RoboDK station: Ensamble.rdk

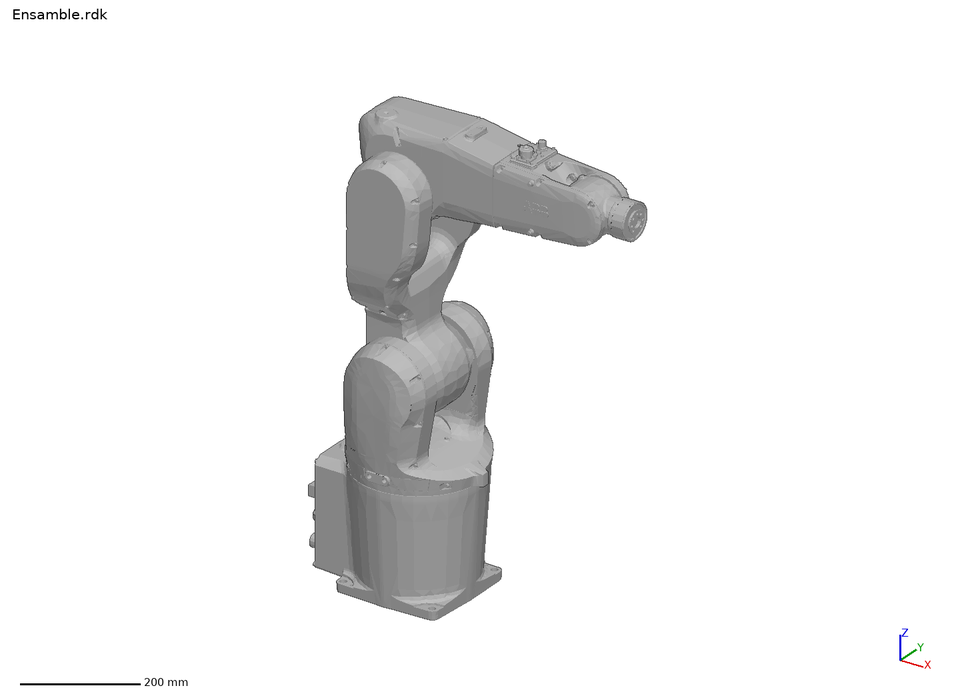
[picture v0: the station drawn from its stored meshes, robots at their saved joint values, targets as dots, program paths as lines]
Station Ensamble (saved by RoboDK 5.3.4). Poses are relative to the parent item; angles as X-Y-Z fixed-axis rotations.
  - object robot_irb_1200-7_0_7_01 at (0, 0, 0) mm, rotated rx 90 ry 0 rz 0 deg, size 285.2 x 192.7 x 127.5 mm, geometry from robot_irb_1200-7_0_7_01.STEP
  - object robot_irb_1200-7_0_7_02 at (0, 0, 0) mm, rotated rx 90 ry 0 rz 0 deg, size 5.5 x 44 x 44 mm, geometry from robot_irb_1200-7_0_7_02.STEP
  - object robot_irb_1200-7_0_7_03 at (0, 0, 0) mm, rotated rx 90 ry 0 rz 0 deg, size 311.7 x 234 x 239.1 mm, geometry from robot_irb_1200-7_0_7_03.STEP
  - object robot_irb_1200-7_0_7_04 at (0, 0, 0) mm, rotated rx 90 ry 0 rz 0 deg, size 234.9 x 147.4 x 121.5 mm, geometry from robot_irb_1200-7_0_7_04.STEP
  - object robot_irb_1200-7_0_7_05 at (0, 0, 0) mm, rotated rx 90 ry 0 rz 0 deg, size 155.5 x 499.9 x 235 mm, geometry from robot_irb_1200-7_0_7_05.STEP
  - object robot_irb_1200-7_0_7_06 at (0, 0, 0) mm, rotated rx 90 ry 0 rz 0 deg, size 258.8 x 261.4 x 263.6 mm, geometry from robot_irb_1200-7_0_7_06.STEP
  - object robot_irb_1200-7_0_7_07 at (0, 0, 0) mm, rotated rx 90 ry 0 rz 0 deg, size 142.6 x 95 x 69 mm, geometry from robot_irb_1200-7_0_7_07.STEP
